FUNCTION_BLOCK TcoLoggerConfiguration
VAR_INPUT
END_VAR
VAR_OUTPUT
END_VAR
VAR
	_minimumLevel			: LogLevel := LogLevel.Info;
	
	_sinks					: LogSinkList;
	_enrichers				: LogEnricherList;

	_enrichmentConfig		: TcoLoggerEnrichmentConfiguration(THIS^);
	_sinksConfig			: TcoLoggerSinkConfiguration(THIS^);
END_VAR

METHOD INTERNAL AddEnrichment : BOOL
VAR_INPUT
	Enricher		: ITcoLogEnricher;
END_VAR
AddEnrichment := _enrichers.AddEnricher(Enricher);
END_METHOD

METHOD INTERNAL AddSink : BOOL
VAR_INPUT
	Sink		: ITcoLogSink;
END_VAR
AddSink := _sinks.AddSink(Sink);
END_METHOD

METHOD PUBLIC Build : BOOL
VAR_INPUT
END_VAR
END_METHOD

METHOD PUBLIC Clear : REFERENCE TO TcoLoggerConfiguration
VAR_INPUT
END_VAR
_minimumLevel := LogLevel.Info;

_sinks.Clear();
MEMSET(ADR(_enrichers), 0, SIZEOF(_enrichers));

Clear := THIS^;
END_METHOD

PROPERTY INTERNAL Enrichers : REFERENCE TO LogEnricherList
GET
Enrichers REF= _enrichers;
END_GET
END_PROPERTY

PROPERTY EnrichWith : REFERENCE TO TcoLoggerEnrichmentConfiguration
GET
EnrichWith REF= _enrichmentConfig;
END_GET
END_PROPERTY

PROPERTY PUBLIC Level : LogLevel
GET
Level := _minimumLevel;
END_GET
END_PROPERTY

METHOD PUBLIC MinimumLevel : REFERENCE TO TcoLoggerConfiguration
VAR_INPUT
	Level		: LogLevel;
END_VAR
END_METHOD

METHOD PUBLIC ReadFrom : REFERENCE TO TcoLoggerConfiguration
VAR_INPUT
	FilePath		: STRING(255);
END_VAR
// Read json config file

// json structure example

(*
{
    "MinimumLevel": "Debug",
    "WriteTo": [
      { "Name": "XAE" },
      { "Name": "File", "Args": { "path": "C:/Temp/log.txt" } }
    ],
    "Enrich": [ "Context", "InstancePath", "ProjectName" ]
}
*)
END_METHOD

PROPERTY INTERNAL Sinks : REFERENCE TO LogSinkList
GET
Sinks REF= _sinks;
END_GET
END_PROPERTY

PROPERTY PUBLIC WriteTo : REFERENCE TO TcoLoggerSinkConfiguration
GET
WriteTo REF= _sinksConfig;
END_GET
END_PROPERTY

END_FUNCTION_BLOCK

(* stored: Version 1.1.0.1, ProductVersion 3.1.4024.9
   POU TcoLoggerConfiguration: Id {afb08e83-e8af-0cf3-1dfe-e9fe07bf3f42}, SpecialFunc None
   Method AddEnrichment: Id {c4e3951e-98d3-0a8d-02d3-1f1bb21a287f}
   Method AddSink: Id {1d367e2a-27e5-0a7b-3b2b-50e57591d203}
   Method Build: Id {9941a9e6-f50e-0f99-220e-4e3a9fd4441e}
   Method Clear: Id {30c875c2-0d1d-02f7-1343-6de286f35d98}
   Property Enrichers: Id {5d9cfc22-8894-044f-03cc-b704392b9942}
   Get Get: Id {5d52f7de-93d6-03e7-3ab6-2b80595efb17}
   Property EnrichWith: Id {b8e5166c-9aff-0aac-1013-2881bc3d3c1b}
   Get Get: Id {45ec0d23-eefd-046d-0458-c18e9d04dec3}
   Property Level: Id {8c802460-c66a-0c59-3511-ba2f14565402}
   Get Get: Id {4ec5a105-9f86-08fc-2c5a-0d5c872b7a7b}
   Method MinimumLevel: Id {6328f6cb-9fff-0862-1a07-6b1bf8314155}
   Method ReadFrom: Id {db489568-ded7-0537-2bb3-5ee5d7c09d84}
   Property Sinks: Id {f32a7f22-4212-0803-0fb3-4501ae755fd8}
   Get Get: Id {fb620794-85e5-09e5-1b7d-08165fa78387}
   Property WriteTo: Id {4558ccb3-bc85-03a8-201d-d3561a45e663}
   Get Get: Id {75351e8b-1bd1-05ca-2882-014b7cbeb497} *)
